TYPE AX5000_P_0100 :
STRUCT
	ASM_nominal_speed:UDINT;
END_STRUCT
END_TYPE

(* stored: Version 1.1.0.1, ProductVersion 3.1.4024.3
   DUT AX5000_P_0100: Id {aa33513c-9913-42fb-9514-689a0598ac72} *)
